% RSLogix 500 project I2A- JOB 11- MITCH_BAK027.RSS, saved by version 10.00.00.00 %
PROJECT "ML01B"    % processor: Bul.1763 MicroLogix 1100 Series B %

PROGRAM FILES
  LAD 2   8 rungs

DATA FILES
  O0 OUTPUT  4 elements
  I1 INPUT  6 elements
  S2 STATUS  66 elements
  B3 BINARY  1 elements
  T4 TIMER  1 elements
  C5 COUNTER  1 elements
  R6 CONTROL  1 elements
  N7 INTEGER  1 elements
  F8 FLOAT  1 elements

LADDER 2
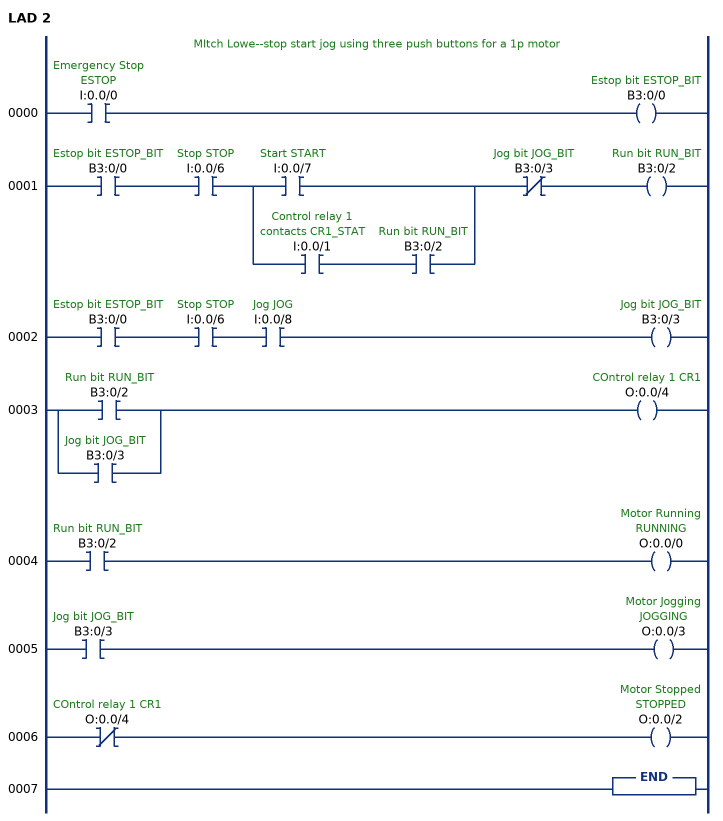
% Rung: 0 %
% MItch Lowe--stop start jog using three push buttons for a 1p motor %
SOR XIC I:0.0/0 OTE B3:0/0 EOR
%   I:0.0/0  ESTOP  "Emergency Stop" %
%   B3:0/0  ESTOP_BIT  "Estop bit" %
% Rung: 1 %
SOR XIC B3:0/0 XIC I:0.0/6 BST XIC I:0.0/7 NXB XIC I:0.0/1 XIC B3:0/2 BND XIO B3:0/3 OTE B3:0/2 EOR
%   B3:0/0  ESTOP_BIT  "Estop bit" %
%   I:0.0/6  STOP  "Stop" %
%   I:0.0/7  START  "Start" %
%   I:0.0/1  CR1_STAT  "Control relay 1 contacts" %
%   B3:0/2  RUN_BIT  "Run bit" %
%   B3:0/3  JOG_BIT  "Jog bit" %
% Rung: 2 %
SOR XIC B3:0/0 XIC I:0.0/6 XIC I:0.0/8 OTE B3:0/3 EOR
%   B3:0/0  ESTOP_BIT  "Estop bit" %
%   I:0.0/6  STOP  "Stop" %
%   I:0.0/8  JOG  "Jog" %
%   B3:0/3  JOG_BIT  "Jog bit" %
% Rung: 3 %
SOR BST XIC B3:0/2 NXB XIC B3:0/3 BND OTE O:0.0/4 EOR
%   B3:0/2  RUN_BIT  "Run bit" %
%   B3:0/3  JOG_BIT  "Jog bit" %
%   O:0.0/4  CR1  "COntrol relay 1" %
% Rung: 4 %
SOR XIC B3:0/2 OTE O:0.0/0 EOR
%   B3:0/2  RUN_BIT  "Run bit" %
%   O:0.0/0  RUNNING  "Motor Running" %
% Rung: 5 %
SOR XIC B3:0/3 OTE O:0.0/3 EOR
%   B3:0/3  JOG_BIT  "Jog bit" %
%   O:0.0/3  JOGGING  "Motor Jogging" %
% Rung: 6 %
SOR XIO O:0.0/4 OTE O:0.0/2 EOR
%   O:0.0/4  CR1  "COntrol relay 1" %
%   O:0.0/2  STOPPED  "Motor Stopped" %
% Rung: 7 %
SOR END EOR

OTHER DOCUMENTED ADDRESSES
  I:0.0/2  CR2_STAT  "Control relay 2 contacts"
  I:0.0/3  3PSSA  "thre position switch A"
  I:0.0/4  3PSS_B  "Three posision selector switch B"
  I:0.0/5  2PSSA  "2 position selector switch A"
  O:0.0/1  YELLOWLT
  O:0.0/5  CR2  "Control relay 2"

DATA TABLE (non-zero values as saved)
DATA B3
% B3:0 % 0X0001
